// TIA Portal V20 export
DATA_BLOCK "instFB_ConveyorCtrl"   // DB
TITLE = instFB_ConveyorCtrl (infeed modularisation, 2026-05-20)
VERSION : 1.1
// Instance DB for FB_ConveyorCtrl (2026-05-20). Owns the palletizing infeed -- SpawnContainerCmd pulse + BeltVelocity belt latch. No MC instances, so zero OB91 (MC-Servo) impact. DB number omitted -- TIA auto-assigns.
// stored: InstanceOfName FB_ConveyorCtrl, InstanceOfType FB
"FB_ConveyorCtrl"
   // VAR
   //    sRTRIGStart { S7_SetPoint := 'True'} : R_TRIG;
   //    sRTRIGStop { S7_SetPoint := 'True'} : R_TRIG;
   //    sRTRIGPacking { S7_SetPoint := 'True'} : R_TRIG;
   //    sRTRIGPalletizing { S7_SetPoint := 'True'} : R_TRIG;
   //    sFTRIGPalletizing { S7_SetPoint := 'True'} : F_TRIG;
   //    sRTRIGSpawnFire { S7_SetPoint := 'True'} : R_TRIG;
   //    instSpawnTimer { S7_SetPoint := 'True'} : TON_TIME;
   //    statRunning : Bool;
   //    statSpawnFire : Bool;
   //    statSpawnActive : Bool;
   //    statBeltRun : Bool;
   //    statSpawnCount : Int;
   // END_VAR
BEGIN
END_DATA_BLOCK
